KUKA KRL program: test4move.src

&ACCESS RVP
&REL 6
&PARAM DISKPATH = KRC:\R1\Program
DEF test4move()

DECL FRAME POS_TEST

BAS(#INITMOV, 0)
PTP $POS_ACT

POS_TEST.Z = $POS_ACT.Z + 10

$VEL.CP=0.9
$VEL.ORI1=5
$VEL.ORI2=5

$APO.CVEL=30
$APO.CDIS=20
LIN POS_TEST C_VEL

END
